RoboDK station: station.rdk

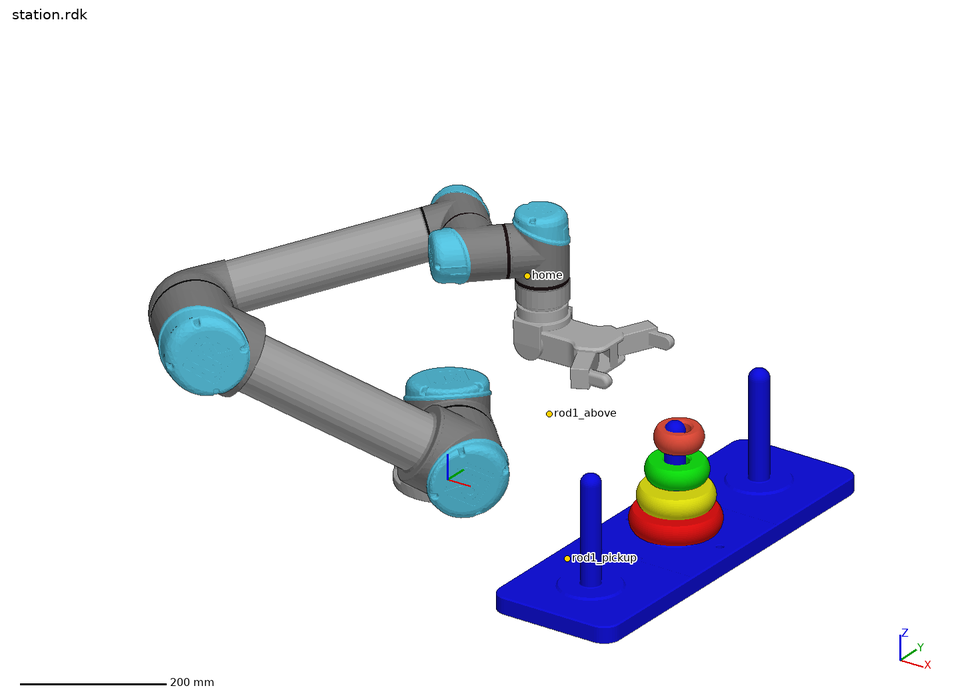
[picture v0: the station drawn from its stored meshes, robots at their saved joint values, targets as dots, program paths as lines]
Station station (saved by RoboDK 5.7.3). Poses are relative to the parent item; angles as X-Y-Z fixed-axis rotations.
  - object base at (380, 1000, -24) mm, rotated rx 90 ry 0 rz 90 deg, size 600.8 x 195 x 200 mm, geometry from base.STL
  - frame UR5 Base at (0, 1000, -40) mm
    - robot UR5: 6 axes
        modified DH rows (alpha deg, a mm, theta deg, d mm): 0, 0, 0, 89.2; 90, 0, 180, 0; 0, 425, 0, 0; 0, 392, 0, 109.3; -90, 0, 0, 94.75; 90, 0, 180, 82.5
        joint limits [-360, -360, -360, -360, -360, -360] to [360, 360, 360, 360, 360, 360]; home [0, -90, -90, 0, 90, 0]; saved at [44.067, -31.007, -136.324, -101.775, 89.133, 44.06]
      - tool tool, TCP at (0, -150, 50) mm, rotated rx 90 ry 0 rz 0 deg, size 203.2 x 72 x 184.8 mm, geometry from tool.STL
    - target home (Cartesian target) at (203.8, -100.26, 406.14) mm, rotated rx -88.75 ry 0 rz -90 deg; joints [13.311, -28.081, -113.408, -127.298, 89.713, 13.308] of UR5
    - target rod1_above (Cartesian target) at (310, -200, 266.38) mm, rotated rx -88.75 ry 0 rz -90 deg; joints [-26.391, -53.049, -132.087, -83.748, 90.553, -26.385] of UR5
    - target rod1_pickup (Cartesian target) at (339.62, -200, 54.03) mm, rotated rx -98.68 ry 0 rz -90 deg; joints [-21.358, -76.91, -149.131, -52.048, 86.85, -21.134] of UR5
  - object disk_130 at (380.76, 1000, 8.94) mm, rotated rx 90 ry 0 rz 0 deg, size 130 x 30 x 130 mm, geometry from 130.STL
  - object disk_110 at (381.51, 1000, 43.88) mm, rotated rx 90 ry 0 rz 0 deg, size 109.9 x 30 x 109.9 mm, geometry from 110.STL
  - object disk_90 at (383.02, 1000, 83.77) mm, rotated rx 90 ry 0 rz 0 deg, size 89.9 x 30 x 89.9 mm, geometry from 90.STL
  - object disk_70 at (386.04, 1000, 133.54) mm, rotated rx 90 ry 0 rz 0 deg, size 70 x 30 x 70 mm, geometry from 70.STL
